SUBAPPLICATION GreenRedBackground2SC (* Hintergrundfarbe (TRUE -> Grün, FALSE -> Rot) für 2 Objekte (Kompakt) *)
  (* Standard: 61499-2 *)
  (* Version 1.0, 2026-07-21, franz, Meisterschulen am Ostbahnhof *)
  PACKAGE MyLib::sys;
  IMPORT isobus::UT::Q::types::s2ObjectIDs;
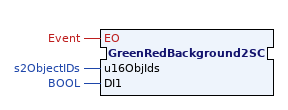
  EVENT_INPUT
    EO;
  END_EVENT
  VAR_INPUT
    u16ObjIds : isobus::UT::Q::types::s2ObjectIDs;
    DI1 : BOOL; (* Selector *)
  END_VAR
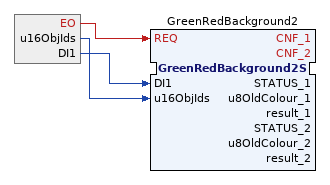
  SUBAPPS
    GreenRedBackground2 : MyLib::sys::GreenRedBackground2S;
  END_SUBAPPS
  EVENT_CONNECTIONS
    EO TO GreenRedBackground2.REQ;
  END_CONNECTIONS
  DATA_CONNECTIONS
    u16ObjIds TO GreenRedBackground2.u16ObjIds;
    DI1 TO GreenRedBackground2.DI1;
  END_CONNECTIONS
END_SUBAPPLICATION
